(* IEC 61131-3 sources: plc_generation_empirical_study/datasets/task_bank_v0_3_1/tasks/C06_B06_composite, 2 files *)

(* ---- interface.st ---- *)
FUNCTION_BLOCK C06_B06_composite
VAR_INPUT
    A_Inspected : BOOL;
    A_Rejected : BOOL;
    A_Reset : BOOL;
    A_WindowSize : INT;
    A_RejectLimit : INT;
    B_Item : BOOL;
    B_Reset : BOOL;
    B_Target : INT;
    B_Enable : BOOL;
    SubsystemBEnable : BOOL;
    CrossReset : BOOL;
END_VAR
VAR_OUTPUT
    A_WindowCount : INT;
    A_RejectCount : INT;
    A_LockedOut : BOOL;
    A_WindowComplete : BOOL;
    B_Count : INT;
    B_BatchDone : BOOL;
    B_Accepted : BOOL;
    CrossReady : BOOL;
    CrossBlocked : BOOL;
END_VAR
END_FUNCTION_BLOCK

(* ---- reference.st ---- *)
FUNCTION_BLOCK C06_B06_composite
VAR_INPUT
    A_Inspected : BOOL;
    A_Rejected : BOOL;
    A_Reset : BOOL;
    A_WindowSize : INT;
    A_RejectLimit : INT;
    B_Item : BOOL;
    B_Reset : BOOL;
    B_Target : INT;
    B_Enable : BOOL;
    SubsystemBEnable : BOOL;
    CrossReset : BOOL;
END_VAR
VAR_OUTPUT
    A_WindowCount : INT;
    A_RejectCount : INT;
    A_LockedOut : BOOL;
    A_WindowComplete : BOOL;
    B_Count : INT;
    B_BatchDone : BOOL;
    B_Accepted : BOOL;
    CrossReady : BOOL;
    CrossBlocked : BOOL;
END_VAR
VAR
    A_PrevInspected : BOOL := FALSE;
    B_PrevItem : BOOL := FALSE;
END_VAR

A_WindowComplete := FALSE;
IF A_Reset THEN
    A_WindowCount := 0;
    A_RejectCount := 0;
    A_LockedOut := FALSE;
ELSIF (NOT A_LockedOut) AND A_Inspected AND (NOT A_PrevInspected) THEN
    A_WindowCount := A_WindowCount + 1;
    IF A_Rejected THEN
        A_RejectCount := A_RejectCount + 1;
    END_IF;
    IF A_WindowCount >= A_WindowSize THEN
        IF A_RejectCount > A_RejectLimit THEN
            A_LockedOut := TRUE;
        END_IF;
        A_WindowCount := 0;
        A_RejectCount := 0;
        A_WindowComplete := TRUE;
    END_IF;
END_IF;
A_PrevInspected := A_Inspected;

IF CrossReset THEN
    CrossReady := FALSE;
ELSIF A_LockedOut THEN
    CrossReady := TRUE;
END_IF;
CrossBlocked := SubsystemBEnable AND (NOT CrossReady);

IF SubsystemBEnable AND CrossReady THEN
    B_Accepted := FALSE;
    IF B_Reset THEN
        B_Count := 0;
    ELSIF B_Enable AND B_Item AND (NOT B_PrevItem) AND (B_Count < B_Target) THEN
        B_Count := B_Count + 1;
        B_Accepted := TRUE;
    END_IF;
    B_BatchDone := B_Count >= B_Target;
    B_PrevItem := B_Item;
ELSE
    B_Count := 0;
    B_BatchDone := FALSE;
    B_Accepted := FALSE;
END_IF;

END_FUNCTION_BLOCK
